(* IEC 61131-3 sources: CodesysTest/alpha/export/FBs/Components/Paper/PerfBreaker.pou, 3 files *)

(* ---- PerfBreaker.pou.st ---- *)
(*#-#-#-#-#-#-#-#-#-#---Declaration---#-#-#-#-#-#-#-#-#-#-#-#-#*)

FUNCTION_BLOCK PerfBreaker EXTENDS FB_ThreePositionCylinder
VAR_INPUT
	upStatusDelay : TIME := T#250MS;
	downStatusDelay : TIME := T#250ms;
END_VAR
VAR_OUTPUT
END_VAR
VAR
	upStatusTimer : TON;
	downStatusTimer : TON;
END_VAR
(*#-#-#-#-#-#-#-#-#-#---Implementation---#-#-#-#-#-#-#-#-#-#-#-#-#*)

//Retract = up, extend = down
upStatusTimer(IN := retractOutput, PT := upStatusDelay);
downStatusTimer(IN := extendOutput, PT := downStatusDelay);
extendedStatus := downStatusTimer.Q;
retractedStatus := upStatusTimer.Q;

(* ---- MoveDown.m.st ---- *)
(*#-#-#-#-#-#-#-#-#-#---Declaration---#-#-#-#-#-#-#-#-#-#-#-#-#*)

METHOD MoveDown
VAR_INPUT
END_VAR
(*#-#-#-#-#-#-#-#-#-#---Implementation---#-#-#-#-#-#-#-#-#-#-#-#-#*)

Extend();

(* ---- MoveUp.m.st ---- *)
(*#-#-#-#-#-#-#-#-#-#---Declaration---#-#-#-#-#-#-#-#-#-#-#-#-#*)

METHOD MoveUp
VAR_INPUT
END_VAR
(*#-#-#-#-#-#-#-#-#-#---Implementation---#-#-#-#-#-#-#-#-#-#-#-#-#*)

Retract();
